{attribute 'GeneratedUsingTerminal: EL2521--0000'}
{attribute addProperty BoxType "EL2521--0000"}
{attribute addProperty Id "StatusAT %I*UINT2Data_InAT %I*UINT2"}
{attribute addProperty CRC "2738050084"}
{attribute addProperty Size "4"}
TYPE Inputs_A3335424 EXTENDS InputBase_8311D824 :
STRUCT
	{attribute addProperty Name "Status"}
	Status AT %I* : UINT;
	{attribute addProperty Name "Data_In"}
	Data_In AT %I* : UINT;
END_STRUCT
END_TYPE

(* stored: Version 1.2.0.0, ProductVersion 3.1.4024.9
   DUT Inputs_A3335424: Id {22371145-c025-4743-bbfe-9b116196ed43} *)
